        state1.dvar_M_South_SCADA := elit_Active;
        IF (("DB".state0.dvar_M_sup_South_Commands) = (elit_NoCommand)) THEN
            state1.dvar_M_sup_South_Commands := elit_DownstreamPaddleStop;
        ELSIF (("DB".state0.dvar_M_sup_South_Commands) = (elit_DownstreamGateOpen)) THEN
            state1.dvar_M_sup_South_Commands := elit_DownstreamGateOpen;
        ELSIF (("DB".state0.dvar_M_sup_South_Commands) = (elit_DownstreamGateClose)) THEN
            state1.dvar_M_sup_South_Commands := elit_DownstreamGateClose;
        ELSIF (("DB".state0.dvar_M_sup_South_Commands) = (elit_DownstreamGateStop)) THEN
            state1.dvar_M_sup_South_Commands := elit_DownstreamGateStop;
        ELSIF (("DB".state0.dvar_M_sup_South_Commands) = (elit_DownstreamPaddleOpen)) THEN
            state1.dvar_M_sup_South_Commands := elit_DownstreamPaddleOpen;
        ELSIF (("DB".state0.dvar_M_sup_South_Commands) = (elit_DownstreamPaddleClose)) THEN
            state1.dvar_M_sup_South_Commands := elit_DownstreamPaddleClose;
        ELSIF (("DB".state0.dvar_M_sup_South_Commands) = (elit_DownstreamPaddleStop)) THEN
            state1.dvar_M_sup_South_Commands := elit_DownstreamPaddleStop;
        ELSIF (("DB".state0.dvar_M_sup_South_Commands) = (elit_DownstreamEnteringTLRedRed)) THEN
            state1.dvar_M_sup_South_Commands := elit_DownstreamEnteringTLRedRed;
        ELSIF (("DB".state0.dvar_M_sup_South_Commands) = (elit_DownstreamEnteringTLRed)) THEN
            state1.dvar_M_sup_South_Commands := elit_DownstreamEnteringTLRed;
        ELSIF (("DB".state0.dvar_M_sup_South_Commands) = (elit_DownstreamEnteringTLRedGreen)) THEN
            state1.dvar_M_sup_South_Commands := elit_DownstreamEnteringTLRedGreen;
        ELSIF (("DB".state0.dvar_M_sup_South_Commands) = (elit_DownstreamEnteringTLGreen)) THEN
            state1.dvar_M_sup_South_Commands := elit_DownstreamEnteringTLGreen;
        ELSIF (("DB".state0.dvar_M_sup_South_Commands) = (elit_DownstreamLeavingTLRed)) THEN
            state1.dvar_M_sup_South_Commands := elit_DownstreamLeavingTLRed;
        ELSIF (("DB".state0.dvar_M_sup_South_Commands) = (elit_DownstreamLeavingTLGreen)) THEN
            state1.dvar_M_sup_South_Commands := elit_DownstreamLeavingTLGreen;
        ELSIF (("DB".state0.dvar_M_sup_South_Commands) = (elit_UpstreamGateOpen)) THEN
            state1.dvar_M_sup_South_Commands := elit_UpstreamGateOpen;
        ELSIF (("DB".state0.dvar_M_sup_South_Commands) = (elit_UpstreamGateClose)) THEN
            state1.dvar_M_sup_South_Commands := elit_UpstreamGateClose;
        ELSIF (("DB".state0.dvar_M_sup_South_Commands) = (elit_UpstreamGateStop)) THEN
            state1.dvar_M_sup_South_Commands := elit_UpstreamGateStop;
        ELSIF (("DB".state0.dvar_M_sup_South_Commands) = (elit_UpstreamPaddleOpen)) THEN
            state1.dvar_M_sup_South_Commands := elit_UpstreamPaddleOpen;
        ELSIF (("DB".state0.dvar_M_sup_South_Commands) = (elit_UpstreamPaddleClose)) THEN
            state1.dvar_M_sup_South_Commands := elit_UpstreamPaddleClose;
        ELSIF (("DB".state0.dvar_M_sup_South_Commands) = (elit_UpstreamPaddleStop)) THEN
            state1.dvar_M_sup_South_Commands := elit_UpstreamPaddleStop;
        ELSIF (("DB".state0.dvar_M_sup_South_Commands) = (elit_UpstreamEnteringTLRedRed)) THEN
            state1.dvar_M_sup_South_Commands := elit_UpstreamEnteringTLRedRed;
        ELSIF (("DB".state0.dvar_M_sup_South_Commands) = (elit_UpstreamEnteringTLRed)) THEN
            state1.dvar_M_sup_South_Commands := elit_UpstreamEnteringTLRed;
        ELSIF (("DB".state0.dvar_M_sup_South_Commands) = (elit_UpstreamEnteringTLRedGreen)) THEN
            state1.dvar_M_sup_South_Commands := elit_UpstreamEnteringTLRedGreen;
        ELSIF (("DB".state0.dvar_M_sup_South_Commands) = (elit_UpstreamEnteringTLGreen)) THEN
            state1.dvar_M_sup_South_Commands := elit_UpstreamEnteringTLGreen;
        ELSIF (("DB".state0.dvar_M_sup_South_Commands) = (elit_UpstreamLeavingTLRed)) THEN
            state1.dvar_M_sup_South_Commands := elit_UpstreamLeavingTLRed;
        ELSIF (("DB".state0.dvar_M_sup_South_Commands) = (elit_UpstreamLeavingTLGreen)) THEN
            state1.dvar_M_sup_South_Commands := elit_UpstreamLeavingTLGreen;
        END_IF;

        "DB".state0 := state1;
    END_IF;
END_IF;

// Event "South_Commands_UpstreamEnteringTLGreen_act".
IF NOT progress THEN
    b1 := ("DB".state0.dvar_M_South_SCADA) = (elit_Inactive);
    b1 := b1 AND ("SCADA".dvar_M_South_SCADA_UpstreamEnteringTLGreen);
    IF b1 THEN
        progress := TRUE;
        state1 := "DB".state0;

        state1.dvar_M_South_SCADA := elit_Active;
        IF (("DB".state0.dvar_M_sup_South_Commands) = (elit_NoCommand)) THEN
            state1.dvar_M_sup_South_Commands := elit_UpstreamEnteringTLGreen;
        ELSIF (("DB".state0.dvar_M_sup_South_Commands) = (elit_DownstreamGateOpen)) THEN
            state1.dvar_M_sup_South_Commands := elit_DownstreamGateOpen;
        ELSIF (("DB".state0.dvar_M_sup_South_Commands) = (elit_DownstreamGateClose)) THEN
            state1.dvar_M_sup_South_Commands := elit_DownstreamGateClose;
        ELSIF (("DB".state0.dvar_M_sup_South_Commands) = (elit_DownstreamGateStop)) THEN
            state1.dvar_M_sup_South_Commands := elit_DownstreamGateStop;
        ELSIF (("DB".state0.dvar_M_sup_South_Commands) = (elit_DownstreamPaddleOpen)) THEN
            state1.dvar_M_sup_South_Commands := elit_DownstreamPaddleOpen;
        ELSIF (("DB".state0.dvar_M_sup_South_Commands) = (elit_DownstreamPaddleClose)) THEN
            state1.dvar_M_sup_South_Commands := elit_DownstreamPaddleClose;
        ELSIF (("DB".state0.dvar_M_sup_South_Commands) = (elit_DownstreamPaddleStop)) THEN
            state1.dvar_M_sup_South_Commands := elit_DownstreamPaddleStop;
        ELSIF (("DB".state0.dvar_M_sup_South_Commands) = (elit_DownstreamEnteringTLRedRed)) THEN
            state1.dvar_M_sup_South_Commands := elit_DownstreamEnteringTLRedRed;
        ELSIF (("DB".state0.dvar_M_sup_South_Commands) = (elit_DownstreamEnteringTLRed)) THEN
            state1.dvar_M_sup_South_Commands := elit_DownstreamEnteringTLRed;
        ELSIF (("DB".state0.dvar_M_sup_South_Commands) = (elit_DownstreamEnteringTLRedGreen)) THEN
            state1.dvar_M_sup_South_Commands := elit_DownstreamEnteringTLRedGreen;
        ELSIF (("DB".state0.dvar_M_sup_South_Commands) = (elit_DownstreamEnteringTLGreen)) THEN
            state1.dvar_M_sup_South_Commands := elit_DownstreamEnteringTLGreen;
        ELSIF (("DB".state0.dvar_M_sup_South_Commands) = (elit_DownstreamLeavingTLRed)) THEN
            state1.dvar_M_sup_South_Commands := elit_DownstreamLeavingTLRed;
        ELSIF (("DB".state0.dvar_M_sup_South_Commands) = (elit_DownstreamLeavingTLGreen)) THEN
            state1.dvar_M_sup_South_Commands := elit_DownstreamLeavingTLGreen;
        ELSIF (("DB".state0.dvar_M_sup_South_Commands) = (elit_UpstreamGateOpen)) THEN
            state1.dvar_M_sup_South_Commands := elit_UpstreamGateOpen;
        ELSIF (("DB".state0.dvar_M_sup_South_Commands) = (elit_UpstreamGateClose)) THEN
            state1.dvar_M_sup_South_Commands := elit_UpstreamGateClose;
        ELSIF (("DB".state0.dvar_M_sup_South_Commands) = (elit_UpstreamGateStop)) THEN
            state1.dvar_M_sup_South_Commands := elit_UpstreamGateStop;
        ELSIF (("DB".state0.dvar_M_sup_South_Commands) = (elit_UpstreamPaddleOpen)) THEN
            state1.dvar_M_sup_South_Commands := elit_UpstreamPaddleOpen;
        ELSIF (("DB".state0.dvar_M_sup_South_Commands) = (elit_UpstreamPaddleClose)) THEN
            state1.dvar_M_sup_South_Commands := elit_UpstreamPaddleClose;
        ELSIF (("DB".state0.dvar_M_sup_South_Commands) = (elit_UpstreamPaddleStop)) THEN
            state1.dvar_M_sup_South_Commands := elit_UpstreamPaddleStop;
        ELSIF (("DB".state0.dvar_M_sup_South_Commands) = (elit_UpstreamEnteringTLRedRed)) THEN
            state1.dvar_M_sup_South_Commands := elit_UpstreamEnteringTLRedRed;
        ELSIF (("DB".state0.dvar_M_sup_South_Commands) = (elit_UpstreamEnteringTLRed)) THEN
            state1.dvar_M_sup_South_Commands := elit_UpstreamEnteringTLRed;
        ELSIF (("DB".state0.dvar_M_sup_South_Commands) = (elit_UpstreamEnteringTLRedGreen)) THEN
            state1.dvar_M_sup_South_Commands := elit_UpstreamEnteringTLRedGreen;
        ELSIF (("DB".state0.dvar_M_sup_South_Commands) = (elit_UpstreamEnteringTLGreen)) THEN
            state1.dvar_M_sup_South_Commands := elit_UpstreamEnteringTLGreen;
        ELSIF (("DB".state0.dvar_M_sup_South_Commands) = (elit_UpstreamLeavingTLRed)) THEN
            state1.dvar_M_sup_South_Commands := elit_UpstreamLeavingTLRed;
        ELSIF (("DB".state0.dvar_M_sup_South_Commands) = (elit_UpstreamLeavingTLGreen)) THEN
            state1.dvar_M_sup_South_Commands := elit_UpstreamLeavingTLGreen;
        END_IF;

        "DB".state0 := state1;
    END_IF;
END_IF;

// Event "South_Commands_UpstreamEnteringTLRed_act".
IF NOT progress THEN
    b1 := ("DB".state0.dvar_M_South_SCADA) = (elit_Inactive);
    b1 := b1 AND ("SCADA".dvar_M_South_SCADA_UpstreamEnteringTLRed);
    IF b1 THEN
        progress := TRUE;
        state1 := "DB".state0;

        state1.dvar_M_South_SCADA := elit_Active;
        IF (("DB".state0.dvar_M_sup_South_Commands) = (elit_NoCommand)) THEN
            state1.dvar_M_sup_South_Commands := elit_UpstreamEnteringTLRed;
        ELSIF (("DB".state0.dvar_M_sup_South_Commands) = (elit_DownstreamGateOpen)) THEN
            state1.dvar_M_sup_South_Commands := elit_DownstreamGateOpen;
        ELSIF (("DB".state0.dvar_M_sup_South_Commands) = (elit_DownstreamGateClose)) THEN
            state1.dvar_M_sup_South_Commands := elit_DownstreamGateClose;
        ELSIF (("DB".state0.dvar_M_sup_South_Commands) = (elit_DownstreamGateStop)) THEN
            state1.dvar_M_sup_South_Commands := elit_DownstreamGateStop;
        ELSIF (("DB".state0.dvar_M_sup_South_Commands) = (elit_DownstreamPaddleOpen)) THEN
            state1.dvar_M_sup_South_Commands := elit_DownstreamPaddleOpen;
        ELSIF (("DB".state0.dvar_M_sup_South_Commands) = (elit_DownstreamPaddleClose)) THEN
            state1.dvar_M_sup_South_Commands := elit_DownstreamPaddleClose;
        ELSIF (("DB".state0.dvar_M_sup_South_Commands) = (elit_DownstreamPaddleStop)) THEN
            state1.dvar_M_sup_South_Commands := elit_DownstreamPaddleStop;
        ELSIF (("DB".state0.dvar_M_sup_South_Commands) = (elit_DownstreamEnteringTLRedRed)) THEN
            state1.dvar_M_sup_South_Commands := elit_DownstreamEnteringTLRedRed;
        ELSIF (("DB".state0.dvar_M_sup_South_Commands) = (elit_DownstreamEnteringTLRed)) THEN
            state1.dvar_M_sup_South_Commands := elit_DownstreamEnteringTLRed;
        ELSIF (("DB".state0.dvar_M_sup_South_Commands) = (elit_DownstreamEnteringTLRedGreen)) THEN
            state1.dvar_M_sup_South_Commands := elit_DownstreamEnteringTLRedGreen;
        ELSIF (("DB".state0.dvar_M_sup_South_Commands) = (elit_DownstreamEnteringTLGreen)) THEN
            state1.dvar_M_sup_South_Commands := elit_DownstreamEnteringTLGreen;
        ELSIF (("DB".state0.dvar_M_sup_South_Commands) = (elit_DownstreamLeavingTLRed)) THEN
            state1.dvar_M_sup_South_Commands := elit_DownstreamLeavingTLRed;
        ELSIF (("DB".state0.dvar_M_sup_South_Commands) = (elit_DownstreamLeavingTLGreen)) THEN
            state1.dvar_M_sup_South_Commands := elit_DownstreamLeavingTLGreen;
        ELSIF (("DB".state0.dvar_M_sup_South_Commands) = (elit_UpstreamGateOpen)) THEN
            state1.dvar_M_sup_South_Commands := elit_UpstreamGateOpen;
        ELSIF (("DB".state0.dvar_M_sup_South_Commands) = (elit_UpstreamGateClose)) THEN
            state1.dvar_M_sup_South_Commands := elit_UpstreamGateClose;
        ELSIF (("DB".state0.dvar_M_sup_South_Commands) = (elit_UpstreamGateStop)) THEN
            state1.dvar_M_sup_South_Commands := elit_UpstreamGateStop;
        ELSIF (("DB".state0.dvar_M_sup_South_Commands) = (elit_UpstreamPaddleOpen)) THEN
            state1.dvar_M_sup_South_Commands := elit_UpstreamPaddleOpen;
        ELSIF (("DB".state0.dvar_M_sup_South_Commands) = (elit_UpstreamPaddleClose)) THEN
            state1.dvar_M_sup_South_Commands := elit_UpstreamPaddleClose;
        ELSIF (("DB".state0.dvar_M_sup_South_Commands) = (elit_UpstreamPaddleStop)) THEN
            state1.dvar_M_sup_South_Commands := elit_UpstreamPaddleStop;
        ELSIF (("DB".state0.dvar_M_sup_South_Commands) = (elit_UpstreamEnteringTLRedRed)) THEN
            state1.dvar_M_sup_South_Commands := elit_UpstreamEnteringTLRedRed;
        ELSIF (("DB".state0.dvar_M_sup_South_Commands) = (elit_UpstreamEnteringTLRed)) THEN
            state1.dvar_M_sup_South_Commands := elit_UpstreamEnteringTLRed;
        ELSIF (("DB".state0.dvar_M_sup_South_Commands) = (elit_UpstreamEnteringTLRedGreen)) THEN
            state1.dvar_M_sup_South_Commands := elit_UpstreamEnteringTLRedGreen;
        ELSIF (("DB".state0.dvar_M_sup_South_Commands) = (elit_UpstreamEnteringTLGreen)) THEN
            state1.dvar_M_sup_South_Commands := elit_UpstreamEnteringTLGreen;
        ELSIF (("DB".state0.dvar_M_sup_South_Commands) = (elit_UpstreamLeavingTLRed)) THEN
            state1.dvar_M_sup_South_Commands := elit_UpstreamLeavingTLRed;
        ELSIF (("DB".state0.dvar_M_sup_South_Commands) = (elit_UpstreamLeavingTLGreen)) THEN
            state1.dvar_M_sup_South_Commands := elit_UpstreamLeavingTLGreen;
        END_IF;

        "DB".state0 := state1;
    END_IF;
END_IF;

// Event "South_Commands_UpstreamEnteringTLRedGreen_act".
IF NOT progress THEN
    b1 := ("DB".state0.dvar_M_South_SCADA) = (elit_Inactive);
    b1 := b1 AND ("SCADA".dvar_M_South_SCADA_UpstreamEnteringTLRedGreen);
    IF b1 THEN
        progress := TRUE;
        state1 := "DB".state0;

        state1.dvar_M_South_SCADA := elit_Active;
        IF (("DB".state0.dvar_M_sup_South_Commands) = (elit_NoCommand)) THEN
            state1.dvar_M_sup_South_Commands := elit_UpstreamEnteringTLRedGreen;
        ELSIF (("DB".state0.dvar_M_sup_South_Commands) = (elit_DownstreamGateOpen)) THEN
            state1.dvar_M_sup_South_Commands := elit_DownstreamGateOpen;
        ELSIF (("DB".state0.dvar_M_sup_South_Commands) = (elit_DownstreamGateClose)) THEN
            state1.dvar_M_sup_South_Commands := elit_DownstreamGateClose;
        ELSIF (("DB".state0.dvar_M_sup_South_Commands) = (elit_DownstreamGateStop)) THEN
            state1.dvar_M_sup_South_Commands := elit_DownstreamGateStop;
        ELSIF (("DB".state0.dvar_M_sup_South_Commands) = (elit_DownstreamPaddleOpen)) THEN
            state1.dvar_M_sup_South_Commands := elit_DownstreamPaddleOpen;
        ELSIF (("DB".state0.dvar_M_sup_South_Commands) = (elit_DownstreamPaddleClose)) THEN
            state1.dvar_M_sup_South_Commands := elit_DownstreamPaddleClose;
        ELSIF (("DB".state0.dvar_M_sup_South_Commands) = (elit_DownstreamPaddleStop)) THEN
            state1.dvar_M_sup_South_Commands := elit_DownstreamPaddleStop;
        ELSIF (("DB".state0.dvar_M_sup_South_Commands) = (elit_DownstreamEnteringTLRedRed)) THEN
            state1.dvar_M_sup_South_Commands := elit_DownstreamEnteringTLRedRed;
        ELSIF (("DB".state0.dvar_M_sup_South_Commands) = (elit_DownstreamEnteringTLRed)) THEN
            state1.dvar_M_sup_South_Commands := elit_DownstreamEnteringTLRed;
        ELSIF (("DB".state0.dvar_M_sup_South_Commands) = (elit_DownstreamEnteringTLRedGreen)) THEN
            state1.dvar_M_sup_South_Commands := elit_DownstreamEnteringTLRedGreen;
        ELSIF (("DB".state0.dvar_M_sup_South_Commands) = (elit_DownstreamEnteringTLGreen)) THEN
            state1.dvar_M_sup_South_Commands := elit_DownstreamEnteringTLGreen;
        ELSIF (("DB".state0.dvar_M_sup_South_Commands) = (elit_DownstreamLeavingTLRed)) THEN
            state1.dvar_M_sup_South_Commands := elit_DownstreamLeavingTLRed;
        ELSIF (("DB".state0.dvar_M_sup_South_Commands) = (elit_DownstreamLeavingTLGreen)) THEN
            state1.dvar_M_sup_South_Commands := elit_DownstreamLeavingTLGreen;
        ELSIF (("DB".state0.dvar_M_sup_South_Commands) = (elit_UpstreamGateOpen)) THEN
            state1.dvar_M_sup_South_Commands := elit_UpstreamGateOpen;
        ELSIF (("DB".state0.dvar_M_sup_South_Commands) = (elit_UpstreamGateClose)) THEN
            state1.dvar_M_sup_South_Commands := elit_UpstreamGateClose;
        ELSIF (("DB".state0.dvar_M_sup_South_Commands) = (elit_UpstreamGateStop)) THEN
            state1.dvar_M_sup_South_Commands := elit_UpstreamGateStop;
        ELSIF (("DB".state0.dvar_M_sup_South_Commands) = (elit_UpstreamPaddleOpen)) THEN
            state1.dvar_M_sup_South_Commands := elit_UpstreamPaddleOpen;
        ELSIF (("DB".state0.dvar_M_sup_South_Commands) = (elit_UpstreamPaddleClose)) THEN
            state1.dvar_M_sup_South_Commands := elit_UpstreamPaddleClose;
        ELSIF (("DB".state0.dvar_M_sup_South_Commands) = (elit_UpstreamPaddleStop)) THEN
            state1.dvar_M_sup_South_Commands := elit_UpstreamPaddleStop;
        ELSIF (("DB".state0.dvar_M_sup_South_Commands) = (elit_UpstreamEnteringTLRedRed)) THEN
            state1.dvar_M_sup_South_Commands := elit_UpstreamEnteringTLRedRed;
        ELSIF (("DB".state0.dvar_M_sup_South_Commands) = (elit_UpstreamEnteringTLRed)) THEN
            state1.dvar_M_sup_South_Commands := elit_UpstreamEnteringTLRed;
        ELSIF (("DB".state0.dvar_M_sup_South_Commands) = (elit_UpstreamEnteringTLRedGreen)) THEN
            state1.dvar_M_sup_South_Commands := elit_UpstreamEnteringTLRedGreen;
        ELSIF (("DB".state0.dvar_M_sup_South_Commands) = (elit_UpstreamEnteringTLGreen)) THEN
            state1.dvar_M_sup_South_Commands := elit_UpstreamEnteringTLGreen;
        ELSIF (("DB".state0.dvar_M_sup_South_Commands) = (elit_UpstreamLeavingTLRed)) THEN
            state1.dvar_M_sup_South_Commands := elit_UpstreamLeavingTLRed;
        ELSIF (("DB".state0.dvar_M_sup_South_Commands) = (elit_UpstreamLeavingTLGreen)) THEN
            state1.dvar_M_sup_South_Commands := elit_UpstreamLeavingTLGreen;
        END_IF;

        "DB".state0 := state1;
    END_IF;
END_IF;

// Event "South_Commands_UpstreamEnteringTLRedRed_act".
IF NOT progress THEN
    b1 := ("DB".state0.dvar_M_South_SCADA) = (elit_Inactive);
    b1 := b1 AND ("SCADA".dvar_M_South_SCADA_UpstreamEnteringTLRedRed);
    IF b1 THEN
        progress := TRUE;
        state1 := "DB".state0;

        state1.dvar_M_South_SCADA := elit_Active;
        IF (("DB".state0.dvar_M_sup_South_Commands) = (elit_NoCommand)) THEN
            state1.dvar_M_sup_South_Commands := elit_UpstreamEnteringTLRedRed;
        ELSIF (("DB".state0.dvar_M_sup_South_Commands) = (elit_DownstreamGateOpen)) THEN
            state1.dvar_M_sup_South_Commands := elit_DownstreamGateOpen;
        ELSIF (("DB".state0.dvar_M_sup_South_Commands) = (elit_DownstreamGateClose)) THEN
            state1.dvar_M_sup_South_Commands := elit_DownstreamGateClose;
        ELSIF (("DB".state0.dvar_M_sup_South_Commands) = (elit_DownstreamGateStop)) THEN
            state1.dvar_M_sup_South_Commands := elit_DownstreamGateStop;
        ELSIF (("DB".state0.dvar_M_sup_South_Commands) = (elit_DownstreamPaddleOpen)) THEN
            state1.dvar_M_sup_South_Commands := elit_DownstreamPaddleOpen;
        ELSIF (("DB".state0.dvar_M_sup_South_Commands) = (elit_DownstreamPaddleClose)) THEN
            state1.dvar_M_sup_South_Commands := elit_DownstreamPaddleClose;
        ELSIF (("DB".state0.dvar_M_sup_South_Commands) = (elit_DownstreamPaddleStop)) THEN
            state1.dvar_M_sup_South_Commands := elit_DownstreamPaddleStop;
        ELSIF (("DB".state0.dvar_M_sup_South_Commands) = (elit_DownstreamEnteringTLRedRed)) THEN
            state1.dvar_M_sup_South_Commands := elit_DownstreamEnteringTLRedRed;
        ELSIF (("DB".state0.dvar_M_sup_South_Commands) = (elit_DownstreamEnteringTLRed)) THEN
            state1.dvar_M_sup_South_Commands := elit_DownstreamEnteringTLRed;
        ELSIF (("DB".state0.dvar_M_sup_South_Commands) = (elit_DownstreamEnteringTLRedGreen)) THEN
            state1.dvar_M_sup_South_Commands := elit_DownstreamEnteringTLRedGreen;
        ELSIF (("DB".state0.dvar_M_sup_South_Commands) = (elit_DownstreamEnteringTLGreen)) THEN
            state1.dvar_M_sup_South_Commands := elit_DownstreamEnteringTLGreen;
        ELSIF (("DB".state0.dvar_M_sup_South_Commands) = (elit_DownstreamLeavingTLRed)) THEN
            state1.dvar_M_sup_South_Commands := elit_DownstreamLeavingTLRed;
        ELSIF (("DB".state0.dvar_M_sup_South_Commands) = (elit_DownstreamLeavingTLGreen)) THEN
            state1.dvar_M_sup_South_Commands := elit_DownstreamLeavingTLGreen;
        ELSIF (("DB".state0.dvar_M_sup_South_Commands) = (elit_UpstreamGateOpen)) THEN
            state1.dvar_M_sup_South_Commands := elit_UpstreamGateOpen;
        ELSIF (("DB".state0.dvar_M_sup_South_Commands) = (elit_UpstreamGateClose)) THEN
            state1.dvar_M_sup_South_Commands := elit_UpstreamGateClose;
        ELSIF (("DB".state0.dvar_M_sup_South_Commands) = (elit_UpstreamGateStop)) THEN
            state1.dvar_M_sup_South_Commands := elit_UpstreamGateStop;
        ELSIF (("DB".state0.dvar_M_sup_South_Commands) = (elit_UpstreamPaddleOpen)) THEN
            state1.dvar_M_sup_South_Commands := elit_UpstreamPaddleOpen;
        ELSIF (("DB".state0.dvar_M_sup_South_Commands) = (elit_UpstreamPaddleClose)) THEN
            state1.dvar_M_sup_South_Commands := elit_UpstreamPaddleClose;
        ELSIF (("DB".state0.dvar_M_sup_South_Commands) = (elit_UpstreamPaddleStop)) THEN
            state1.dvar_M_sup_South_Commands := elit_UpstreamPaddleStop;
        ELSIF (("DB".state0.dvar_M_sup_South_Commands) = (elit_UpstreamEnteringTLRedRed)) THEN
            state1.dvar_M_sup_South_Commands := elit_UpstreamEnteringTLRedRed;
        ELSIF (("DB".state0.dvar_M_sup_South_Commands) = (elit_UpstreamEnteringTLRed)) THEN
            state1.dvar_M_sup_South_Commands := elit_UpstreamEnteringTLRed;
        ELSIF (("DB".state0.dvar_M_sup_South_Commands) = (elit_UpstreamEnteringTLRedGreen)) THEN
            state1.dvar_M_sup_South_Commands := elit_UpstreamEnteringTLRedGreen;
        ELSIF (("DB".state0.dvar_M_sup_South_Commands) = (elit_UpstreamEnteringTLGreen)) THEN
            state1.dvar_M_sup_South_Commands := elit_UpstreamEnteringTLGreen;
        ELSIF (("DB".state0.dvar_M_sup_South_Commands) = (elit_UpstreamLeavingTLRed)) THEN
            state1.dvar_M_sup_South_Commands := elit_UpstreamLeavingTLRed;
        ELSIF (("DB".state0.dvar_M_sup_South_Commands) = (elit_UpstreamLeavingTLGreen)) THEN
            state1.dvar_M_sup_South_Commands := elit_UpstreamLeavingTLGreen;
        END_IF;

        "DB".state0 := state1;
    END_IF;
END_IF;

// Event "South_Commands_UpstreamGateClose_act".
IF NOT progress THEN
    b1 := ("DB".state0.dvar_M_South_SCADA) = (elit_Inactive);
    b1 := b1 AND ("SCADA".dvar_M_South_SCADA_UpstreamGateClose);
    IF b1 THEN
        progress := TRUE;
        state1 := "DB".state0;

        state1.dvar_M_South_SCADA := elit_Active;
        IF (("DB".state0.dvar_M_sup_South_Commands) = (elit_NoCommand)) THEN
            state1.dvar_M_sup_South_Commands := elit_UpstreamGateClose;
        ELSIF (("DB".state0.dvar_M_sup_South_Commands) = (elit_DownstreamGateOpen)) THEN
            state1.dvar_M_sup_South_Commands := elit_DownstreamGateOpen;
        ELSIF (("DB".state0.dvar_M_sup_South_Commands) = (elit_DownstreamGateClose)) THEN
            state1.dvar_M_sup_South_Commands := elit_DownstreamGateClose;
        ELSIF (("DB".state0.dvar_M_sup_South_Commands) = (elit_DownstreamGateStop)) THEN
            state1.dvar_M_sup_South_Commands := elit_DownstreamGateStop;
        ELSIF (("DB".state0.dvar_M_sup_South_Commands) = (elit_DownstreamPaddleOpen)) THEN
            state1.dvar_M_sup_South_Commands := elit_DownstreamPaddleOpen;
        ELSIF (("DB".state0.dvar_M_sup_South_Commands) = (elit_DownstreamPaddleClose)) THEN
            state1.dvar_M_sup_South_Commands := elit_DownstreamPaddleClose;
        ELSIF (("DB".state0.dvar_M_sup_South_Commands) = (elit_DownstreamPaddleStop)) THEN
            state1.dvar_M_sup_South_Commands := elit_DownstreamPaddleStop;
        ELSIF (("DB".state0.dvar_M_sup_South_Commands) = (elit_DownstreamEnteringTLRedRed)) THEN
            state1.dvar_M_sup_South_Commands := elit_DownstreamEnteringTLRedRed;
        ELSIF (("DB".state0.dvar_M_sup_South_Commands) = (elit_DownstreamEnteringTLRed)) THEN
            state1.dvar_M_sup_South_Commands := elit_DownstreamEnteringTLRed;
        ELSIF (("DB".state0.dvar_M_sup_South_Commands) = (elit_DownstreamEnteringTLRedGreen)) THEN
            state1.dvar_M_sup_South_Commands := elit_DownstreamEnteringTLRedGreen;
        ELSIF (("DB".state0.dvar_M_sup_South_Commands) = (elit_DownstreamEnteringTLGreen)) THEN
            state1.dvar_M_sup_South_Commands := elit_DownstreamEnteringTLGreen;
        ELSIF (("DB".state0.dvar_M_sup_South_Commands) = (elit_DownstreamLeavingTLRed)) THEN
            state1.dvar_M_sup_South_Commands := elit_DownstreamLeavingTLRed;
        ELSIF (("DB".state0.dvar_M_sup_South_Commands) = (elit_DownstreamLeavingTLGreen)) THEN
            state1.dvar_M_sup_South_Commands := elit_DownstreamLeavingTLGreen;
        ELSIF (("DB".state0.dvar_M_sup_South_Commands) = (elit_UpstreamGateOpen)) THEN
            state1.dvar_M_sup_South_Commands := elit_UpstreamGateOpen;
        ELSIF (("DB".state0.dvar_M_sup_South_Commands) = (elit_UpstreamGateClose)) THEN
            state1.dvar_M_sup_South_Commands := elit_UpstreamGateClose;
        ELSIF (("DB".state0.dvar_M_sup_South_Commands) = (elit_UpstreamGateStop)) THEN
            state1.dvar_M_sup_South_Commands := elit_UpstreamGateStop;
        ELSIF (("DB".state0.dvar_M_sup_South_Commands) = (elit_UpstreamPaddleOpen)) THEN
            state1.dvar_M_sup_South_Commands := elit_UpstreamPaddleOpen;
        ELSIF (("DB".state0.dvar_M_sup_South_Commands) = (elit_UpstreamPaddleClose)) THEN
            state1.dvar_M_sup_South_Commands := elit_UpstreamPaddleClose;
        ELSIF (("DB".state0.dvar_M_sup_South_Commands) = (elit_UpstreamPaddleStop)) THEN
            state1.dvar_M_sup_South_Commands := elit_UpstreamPaddleStop;
        ELSIF (("DB".state0.dvar_M_sup_South_Commands) = (elit_UpstreamEnteringTLRedRed)) THEN
            state1.dvar_M_sup_South_Commands := elit_UpstreamEnteringTLRedRed;
        ELSIF (("DB".state0.dvar_M_sup_South_Commands) = (elit_UpstreamEnteringTLRed)) THEN
            state1.dvar_M_sup_South_Commands := elit_UpstreamEnteringTLRed;
        ELSIF (("DB".state0.dvar_M_sup_South_Commands) = (elit_UpstreamEnteringTLRedGreen)) THEN
            state1.dvar_M_sup_South_Commands := elit_UpstreamEnteringTLRedGreen;
        ELSIF (("DB".state0.dvar_M_sup_South_Commands) = (elit_UpstreamEnteringTLGreen)) THEN
            state1.dvar_M_sup_South_Commands := elit_UpstreamEnteringTLGreen;
        ELSIF (("DB".state0.dvar_M_sup_South_Commands) = (elit_UpstreamLeavingTLRed)) THEN
            state1.dvar_M_sup_South_Commands := elit_UpstreamLeavingTLRed;
        ELSIF (("DB".state0.dvar_M_sup_South_Commands) = (elit_UpstreamLeavingTLGreen)) THEN
            state1.dvar_M_sup_South_Commands := elit_UpstreamLeavingTLGreen;
        END_IF;

        "DB".state0 := state1;
    END_IF;
END_IF;

// Event "South_Commands_UpstreamGateOpen_act".
IF NOT progress THEN
    b1 := ("DB".state0.dvar_M_South_SCADA) = (elit_Inactive);
    b1 := b1 AND ("SCADA".dvar_M_South_SCADA_UpstreamGateOpen);
    IF b1 THEN
        progress := TRUE;
        state1 := "DB".state0;

        state1.dvar_M_South_SCADA := elit_Active;
        IF (("DB".state0.dvar_M_sup_South_Commands) = (elit_NoCommand)) THEN
            state1.dvar_M_sup_South_Commands := elit_UpstreamGateOpen;
        ELSIF (("DB".state0.dvar_M_sup_South_Commands) = (elit_DownstreamGateOpen)) THEN
            state1.dvar_M_sup_South_Commands := elit_DownstreamGateOpen;
        ELSIF (("DB".state0.dvar_M_sup_South_Commands) = (elit_DownstreamGateClose)) THEN
            state1.dvar_M_sup_South_Commands := elit_DownstreamGateClose;
        ELSIF (("DB".state0.dvar_M_sup_South_Commands) = (elit_DownstreamGateStop)) THEN
            state1.dvar_M_sup_South_Commands := elit_DownstreamGateStop;
        ELSIF (("DB".state0.dvar_M_sup_South_Commands) = (elit_DownstreamPaddleOpen)) THEN
            state1.dvar_M_sup_South_Commands := elit_DownstreamPaddleOpen;
        ELSIF (("DB".state0.dvar_M_sup_South_Commands) = (elit_DownstreamPaddleClose)) THEN
            state1.dvar_M_sup_South_Commands := elit_DownstreamPaddleClose;
        ELSIF (("DB".state0.dvar_M_sup_South_Commands) = (elit_DownstreamPaddleStop)) THEN
            state1.dvar_M_sup_South_Commands := elit_DownstreamPaddleStop;
        ELSIF (("DB".state0.dvar_M_sup_South_Commands) = (elit_DownstreamEnteringTLRedRed)) THEN
            state1.dvar_M_sup_South_Commands := elit_DownstreamEnteringTLRedRed;
        ELSIF (("DB".state0.dvar_M_sup_South_Commands) = (elit_DownstreamEnteringTLRed)) THEN
            state1.dvar_M_sup_South_Commands := elit_DownstreamEnteringTLRed;
        ELSIF (("DB".state0.dvar_M_sup_South_Commands) = (elit_DownstreamEnteringTLRedGreen)) THEN
            state1.dvar_M_sup_South_Commands := elit_DownstreamEnteringTLRedGreen;
        ELSIF (("DB".state0.dvar_M_sup_South_Commands) = (elit_DownstreamEnteringTLGreen)) THEN
            state1.dvar_M_sup_South_Commands := elit_DownstreamEnteringTLGreen;
        ELSIF (("DB".state0.dvar_M_sup_South_Commands) = (elit_DownstreamLeavingTLRed)) THEN
            state1.dvar_M_sup_South_Commands := elit_DownstreamLeavingTLRed;
        ELSIF (("DB".state0.dvar_M_sup_South_Commands) = (elit_DownstreamLeavingTLGreen)) THEN
            state1.dvar_M_sup_South_Commands := elit_DownstreamLeavingTLGreen;
        ELSIF (("DB".state0.dvar_M_sup_South_Commands) = (elit_UpstreamGateOpen)) THEN
            state1.dvar_M_sup_South_Commands := elit_UpstreamGateOpen;
        ELSIF (("DB".state0.dvar_M_sup_South_Commands) = (elit_UpstreamGateClose)) THEN
            state1.dvar_M_sup_South_Commands := elit_UpstreamGateClose;
        ELSIF (("DB".state0.dvar_M_sup_South_Commands) = (elit_UpstreamGateStop)) THEN
            state1.dvar_M_sup_South_Commands := elit_UpstreamGateStop;
        ELSIF (("DB".state0.dvar_M_sup_South_Commands) = (elit_UpstreamPaddleOpen)) THEN
            state1.dvar_M_sup_South_Commands := elit_UpstreamPaddleOpen;
        ELSIF (("DB".state0.dvar_M_sup_South_Commands) = (elit_UpstreamPaddleClose)) THEN
            state1.dvar_M_sup_South_Commands := elit_UpstreamPaddleClose;
        ELSIF (("DB".state0.dvar_M_sup_South_Commands) = (elit_UpstreamPaddleStop)) THEN
            state1.dvar_M_sup_South_Commands := elit_UpstreamPaddleStop;
        ELSIF (("DB".state0.dvar_M_sup_South_Commands) = (elit_UpstreamEnteringTLRedRed)) THEN
            state1.dvar_M_sup_South_Commands := elit_UpstreamEnteringTLRedRed;
        ELSIF (("DB".state0.dvar_M_sup_South_Commands) = (elit_UpstreamEnteringTLRed)) THEN
            state1.dvar_M_sup_South_Commands := elit_UpstreamEnteringTLRed;
        ELSIF (("DB".state0.dvar_M_sup_South_Commands) = (elit_UpstreamEnteringTLRedGreen)) THEN
            state1.dvar_M_sup_South_Commands := elit_UpstreamEnteringTLRedGreen;
        ELSIF (("DB".state0.dvar_M_sup_South_Commands) = (elit_UpstreamEnteringTLGreen)) THEN
            state1.dvar_M_sup_South_Commands := elit_UpstreamEnteringTLGreen;
        ELSIF (("DB".state0.dvar_M_sup_South_Commands) = (elit_UpstreamLeavingTLRed)) THEN
            state1.dvar_M_sup_South_Commands := elit_UpstreamLeavingTLRed;
        ELSIF (("DB".state0.dvar_M_sup_South_Commands) = (elit_UpstreamLeavingTLGreen)) THEN
            state1.dvar_M_sup_South_Commands := elit_UpstreamLeavingTLGreen;
        END_IF;

        "DB".state0 := state1;
    END_IF;
END_IF;

// Event "South_Commands_UpstreamGateStop_act".
IF NOT progress THEN
    b1 := ("DB".state0.dvar_M_South_SCADA) = (elit_Inactive);
    b1 := b1 AND ("SCADA".dvar_M_South_SCADA_UpstreamGateStop);
    IF b1 THEN
        progress := TRUE;
        state1 := "DB".state0;

        state1.dvar_M_South_SCADA := elit_Active;
        IF (("DB".state0.dvar_M_sup_South_Commands) = (elit_NoCommand)) THEN
            state1.dvar_M_sup_South_Commands := elit_UpstreamGateStop;
        ELSIF (("DB".state0.dvar_M_sup_South_Commands) = (elit_DownstreamGateOpen)) THEN
            state1.dvar_M_sup_South_Commands := elit_DownstreamGateOpen;
        ELSIF (("DB".state0.dvar_M_sup_South_Commands) = (elit_DownstreamGateClose)) THEN
            state1.dvar_M_sup_South_Commands := elit_DownstreamGateClose;
        ELSIF (("DB".state0.dvar_M_sup_South_Commands) = (elit_DownstreamGateStop)) THEN
            state1.dvar_M_sup_South_Commands := elit_DownstreamGateStop;
        ELSIF (("DB".state0.dvar_M_sup_South_Commands) = (elit_DownstreamPaddleOpen)) THEN
            state1.dvar_M_sup_South_Commands := elit_DownstreamPaddleOpen;
        ELSIF (("DB".state0.dvar_M_sup_South_Commands) = (elit_DownstreamPaddleClose)) THEN
            state1.dvar_M_sup_South_Commands := elit_DownstreamPaddleClose;
        ELSIF (("DB".state0.dvar_M_sup_South_Commands) = (elit_DownstreamPaddleStop)) THEN
            state1.dvar_M_sup_South_Commands := elit_DownstreamPaddleStop;
        ELSIF (("DB".state0.dvar_M_sup_South_Commands) = (elit_DownstreamEnteringTLRedRed)) THEN
            state1.dvar_M_sup_South_Commands := elit_DownstreamEnteringTLRedRed;
        ELSIF (("DB".state0.dvar_M_sup_South_Commands) = (elit_DownstreamEnteringTLRed)) THEN
            state1.dvar_M_sup_South_Commands := elit_DownstreamEnteringTLRed;
        ELSIF (("DB".state0.dvar_M_sup_South_Commands) = (elit_DownstreamEnteringTLRedGreen)) THEN
            state1.dvar_M_sup_South_Commands := elit_DownstreamEnteringTLRedGreen;
        ELSIF (("DB".state0.dvar_M_sup_South_Commands) = (elit_DownstreamEnteringTLGreen)) THEN
            state1.dvar_M_sup_South_Commands := elit_DownstreamEnteringTLGreen;
        ELSIF (("DB".state0.dvar_M_sup_South_Commands) = (elit_DownstreamLeavingTLRed)) THEN
            state1.dvar_M_sup_South_Commands := elit_DownstreamLeavingTLRed;
        ELSIF (("DB".state0.dvar_M_sup_South_Commands) = (elit_DownstreamLeavingTLGreen)) THEN
            state1.dvar_M_sup_South_Commands := elit_DownstreamLeavingTLGreen;
        ELSIF (("DB".state0.dvar_M_sup_South_Commands) = (elit_UpstreamGateOpen)) THEN
            state1.dvar_M_sup_South_Commands := elit_UpstreamGateOpen;
        ELSIF (("DB".state0.dvar_M_sup_South_Commands) = (elit_UpstreamGateClose)) THEN
            state1.dvar_M_sup_South_Commands := elit_UpstreamGateClose;
        ELSIF (("DB".state0.dvar_M_sup_South_Commands) = (elit_UpstreamGateStop)) THEN
            state1.dvar_M_sup_South_Commands := elit_UpstreamGateStop;
        ELSIF (("DB".state0.dvar_M_sup_South_Commands) = (elit_UpstreamPaddleOpen)) THEN
            state1.dvar_M_sup_South_Commands := elit_UpstreamPaddleOpen;
        ELSIF (("DB".state0.dvar_M_sup_South_Commands) = (elit_UpstreamPaddleClose)) THEN
            state1.dvar_M_sup_South_Commands := elit_UpstreamPaddleClose;
        ELSIF (("DB".state0.dvar_M_sup_South_Commands) = (elit_UpstreamPaddleStop)) THEN
            state1.dvar_M_sup_South_Commands := elit_UpstreamPaddleStop;
        ELSIF (("DB".state0.dvar_M_sup_South_Commands) = (elit_UpstreamEnteringTLRedRed)) THEN
            state1.dvar_M_sup_South_Commands := elit_UpstreamEnteringTLRedRed;
        ELSIF (("DB".state0.dvar_M_sup_South_Commands) = (elit_UpstreamEnteringTLRed)) THEN
            state1.dvar_M_sup_South_Commands := elit_UpstreamEnteringTLRed;
        ELSIF (("DB".state0.dvar_M_sup_South_Commands) = (elit_UpstreamEnteringTLRedGreen)) THEN
            state1.dvar_M_sup_South_Commands := elit_UpstreamEnteringTLRedGreen;
        ELSIF (("DB".state0.dvar_M_sup_South_Commands) = (elit_UpstreamEnteringTLGreen)) THEN
            state1.dvar_M_sup_South_Commands := elit_UpstreamEnteringTLGreen;
        ELSIF (("DB".state0.dvar_M_sup_South_Commands) = (elit_UpstreamLeavingTLRed)) THEN
            state1.dvar_M_sup_South_Commands := elit_UpstreamLeavingTLRed;
        ELSIF (("DB".state0.dvar_M_sup_South_Commands) = (elit_UpstreamLeavingTLGreen)) THEN
            state1.dvar_M_sup_South_Commands := elit_UpstreamLeavingTLGreen;
        END_IF;

        "DB".state0 := state1;
    END_IF;
END_IF;

// Event "South_Commands_UpstreamLeavingTLGreen_act".
IF NOT progress THEN
    b1 := ("DB".state0.dvar_M_South_SCADA) = (elit_Inactive);
    b1 := b1 AND ("SCADA".dvar_M_South_SCADA_UpstreamLeavingTLGreen);
    IF b1 THEN
        progress := TRUE;
        state1 := "DB".state0;

        state1.dvar_M_South_SCADA := elit_Active;
        IF (("DB".state0.dvar_M_sup_South_Commands) = (elit_NoCommand)) THEN
            state1.dvar_M_sup_South_Commands := elit_UpstreamLeavingTLGreen;
        ELSIF (("DB".state0.dvar_M_sup_South_Commands) = (elit_DownstreamGateOpen)) THEN
            state1.dvar_M_sup_South_Commands := elit_DownstreamGateOpen;
        ELSIF (("DB".state0.dvar_M_sup_South_Commands) = (elit_DownstreamGateClose)) THEN
            state1.dvar_M_sup_South_Commands := elit_DownstreamGateClose;
        ELSIF (("DB".state0.dvar_M_sup_South_Commands) = (elit_DownstreamGateStop)) THEN
            state1.dvar_M_sup_South_Commands := elit_DownstreamGateStop;
        ELSIF (("DB".state0.dvar_M_sup_South_Commands) = (elit_DownstreamPaddleOpen)) THEN
            state1.dvar_M_sup_South_Commands := elit_DownstreamPaddleOpen;
        ELSIF (("DB".state0.dvar_M_sup_South_Commands) = (elit_DownstreamPaddleClose)) THEN
            state1.dvar_M_sup_South_Commands := elit_DownstreamPaddleClose;
        ELSIF (("DB".state0.dvar_M_sup_South_Commands) = (elit_DownstreamPaddleStop)) THEN
            state1.dvar_M_sup_South_Commands := elit_DownstreamPaddleStop;
        ELSIF (("DB".state0.dvar_M_sup_South_Commands) = (elit_DownstreamEnteringTLRedRed)) THEN
            state1.dvar_M_sup_South_Commands := elit_DownstreamEnteringTLRedRed;
        ELSIF (("DB".state0.dvar_M_sup_South_Commands) = (elit_DownstreamEnteringTLRed)) THEN
            state1.dvar_M_sup_South_Commands := elit_DownstreamEnteringTLRed;
        ELSIF (("DB".state0.dvar_M_sup_South_Commands) = (elit_DownstreamEnteringTLRedGreen)) THEN
            state1.dvar_M_sup_South_Commands := elit_DownstreamEnteringTLRedGreen;
        ELSIF (("DB".state0.dvar_M_sup_South_Commands) = (elit_DownstreamEnteringTLGreen)) THEN
            state1.dvar_M_sup_South_Commands := elit_DownstreamEnteringTLGreen;
        ELSIF (("DB".state0.dvar_M_sup_South_Commands) = (elit_DownstreamLeavingTLRed)) THEN
            state1.dvar_M_sup_South_Commands := elit_DownstreamLeavingTLRed;
        ELSIF (("DB".state0.dvar_M_sup_South_Commands) = (elit_DownstreamLeavingTLGreen)) THEN
            state1.dvar_M_sup_South_Commands := elit_DownstreamLeavingTLGreen;
        ELSIF (("DB".state0.dvar_M_sup_South_Commands) = (elit_UpstreamGateOpen)) THEN
            state1.dvar_M_sup_South_Commands := elit_UpstreamGateOpen;
        ELSIF (("DB".state0.dvar_M_sup_South_Commands) = (elit_UpstreamGateClose)) THEN
            state1.dvar_M_sup_South_Commands := elit_UpstreamGateClose;
        ELSIF (("DB".state0.dvar_M_sup_South_Commands) = (elit_UpstreamGateStop)) THEN
            state1.dvar_M_sup_South_Commands := elit_UpstreamGateStop;
        ELSIF (("DB".state0.dvar_M_sup_South_Commands) = (elit_UpstreamPaddleOpen)) THEN
            state1.dvar_M_sup_South_Commands := elit_UpstreamPaddleOpen;
        ELSIF (("DB".state0.dvar_M_sup_South_Commands) = (elit_UpstreamPaddleClose)) THEN
            state1.dvar_M_sup_South_Commands := elit_UpstreamPaddleClose;
        ELSIF (("DB".state0.dvar_M_sup_South_Commands) = (elit_UpstreamPaddleStop)) THEN
            state1.dvar_M_sup_South_Commands := elit_UpstreamPaddleStop;
        ELSIF (("DB".state0.dvar_M_sup_South_Commands) = (elit_UpstreamEnteringTLRedRed)) THEN
            state1.dvar_M_sup_South_Commands := elit_UpstreamEnteringTLRedRed;
        ELSIF (("DB".state0.dvar_M_sup_South_Commands) = (elit_UpstreamEnteringTLRed)) THEN
            state1.dvar_M_sup_South_Commands := elit_UpstreamEnteringTLRed;
        ELSIF (("DB".state0.dvar_M_sup_South_Commands) = (elit_UpstreamEnteringTLRedGreen)) THEN
            state1.dvar_M_sup_South_Commands := elit_UpstreamEnteringTLRedGreen;
        ELSIF (("DB".state0.dvar_M_sup_South_Commands) = (elit_UpstreamEnteringTLGreen)) THEN
            state1.dvar_M_sup_South_Commands := elit_UpstreamEnteringTLGreen;
        ELSIF (("DB".state0.dvar_M_sup_South_Commands) = (elit_UpstreamLeavingTLRed)) THEN
            state1.dvar_M_sup_South_Commands := elit_UpstreamLeavingTLRed;
        ELSIF (("DB".state0.dvar_M_sup_South_Commands) = (elit_UpstreamLeavingTLGreen)) THEN
            state1.dvar_M_sup_South_Commands := elit_UpstreamLeavingTLGreen;
        END_IF;

        "DB".state0 := state1;
    END_IF;
END_IF;

// Event "South_Commands_UpstreamLeavingTLRed_act".
IF NOT progress THEN
    b1 := ("DB".state0.dvar_M_South_SCADA) = (elit_Inactive);
    b1 := b1 AND ("SCADA".dvar_M_South_SCADA_UpstreamLeavingTLRed);
    IF b1 THEN
        progress := TRUE;
        state1 := "DB".state0;

        state1.dvar_M_South_SCADA := elit_Active;
        IF (("DB".state0.dvar_M_sup_South_Commands) = (elit_NoCommand)) THEN
            state1.dvar_M_sup_South_Commands := elit_UpstreamLeavingTLRed;
        ELSIF (("DB".state0.dvar_M_sup_South_Commands) = (elit_DownstreamGateOpen)) THEN
            state1.dvar_M_sup_South_Commands := elit_DownstreamGateOpen;
        ELSIF (("DB".state0.dvar_M_sup_South_Commands) = (elit_DownstreamGateClose)) THEN
            state1.dvar_M_sup_South_Commands := elit_DownstreamGateClose;
        ELSIF (("DB".state0.dvar_M_sup_South_Commands) = (elit_DownstreamGateStop)) THEN
            state1.dvar_M_sup_South_Commands := elit_DownstreamGateStop;
        ELSIF (("DB".state0.dvar_M_sup_South_Commands) = (elit_DownstreamPaddleOpen)) THEN
            state1.dvar_M_sup_South_Commands := elit_DownstreamPaddleOpen;
        ELSIF (("DB".state0.dvar_M_sup_South_Commands) = (elit_DownstreamPaddleClose)) THEN
            state1.dvar_M_sup_South_Commands := elit_DownstreamPaddleClose;
        ELSIF (("DB".state0.dvar_M_sup_South_Commands) = (elit_DownstreamPaddleStop)) THEN
            state1.dvar_M_sup_South_Commands := elit_DownstreamPaddleStop;
        ELSIF (("DB".state0.dvar_M_sup_South_Commands) = (elit_DownstreamEnteringTLRedRed)) THEN
            state1.dvar_M_sup_South_Commands := elit_DownstreamEnteringTLRedRed;
        ELSIF (("DB".state0.dvar_M_sup_South_Commands) = (elit_DownstreamEnteringTLRed)) THEN
            state1.dvar_M_sup_South_Commands := elit_DownstreamEnteringTLRed;
        ELSIF (("DB".state0.dvar_M_sup_South_Commands) = (elit_DownstreamEnteringTLRedGreen)) THEN
            state1.dvar_M_sup_South_Commands := elit_DownstreamEnteringTLRedGreen;
        ELSIF (("DB".state0.dvar_M_sup_South_Commands) = (elit_DownstreamEnteringTLGreen)) THEN
            state1.dvar_M_sup_South_Commands := elit_DownstreamEnteringTLGreen;
        ELSIF (("DB".state0.dvar_M_sup_South_Commands) = (elit_DownstreamLeavingTLRed)) THEN
            state1.dvar_M_sup_South_Commands := elit_DownstreamLeavingTLRed;
        ELSIF (("DB".state0.dvar_M_sup_South_Commands) = (elit_DownstreamLeavingTLGreen)) THEN
            state1.dvar_M_sup_South_Commands := elit_DownstreamLeavingTLGreen;
        ELSIF (("DB".state0.dvar_M_sup_South_Commands) = (elit_UpstreamGateOpen)) THEN
            state1.dvar_M_sup_South_Commands := elit_UpstreamGateOpen;
        ELSIF (("DB".state0.dvar_M_sup_South_Commands) = (elit_UpstreamGateClose)) THEN
            state1.dvar_M_sup_South_Commands := elit_UpstreamGateClose;
        ELSIF (("DB".state0.dvar_M_sup_South_Commands) = (elit_UpstreamGateStop)) THEN
            state1.dvar_M_sup_South_Commands := elit_UpstreamGateStop;
        ELSIF (("DB".state0.dvar_M_sup_South_Commands) = (elit_UpstreamPaddleOpen)) THEN
            state1.dvar_M_sup_South_Commands := elit_UpstreamPaddleOpen;
        ELSIF (("DB".state0.dvar_M_sup_South_Commands) = (elit_UpstreamPaddleClose)) THEN
            state1.dvar_M_sup_South_Commands := elit_UpstreamPaddleClose;
        ELSIF (("DB".state0.dvar_M_sup_South_Commands) = (elit_UpstreamPaddleStop)) THEN
            state1.dvar_M_sup_South_Commands := elit_UpstreamPaddleStop;
        ELSIF (("DB".state0.dvar_M_sup_South_Commands) = (elit_UpstreamEnteringTLRedRed)) THEN
            state1.dvar_M_sup_South_Commands := elit_UpstreamEnteringTLRedRed;
        ELSIF (("DB".state0.dvar_M_sup_South_Commands) = (elit_UpstreamEnteringTLRed)) THEN
            state1.dvar_M_sup_South_Commands := elit_UpstreamEnteringTLRed;
        ELSIF (("DB".state0.dvar_M_sup_South_Commands) = (elit_UpstreamEnteringTLRedGreen)) THEN
            state1.dvar_M_sup_South_Commands := elit_UpstreamEnteringTLRedGreen;
        ELSIF (("DB".state0.dvar_M_sup_South_Commands) = (elit_UpstreamEnteringTLGreen)) THEN
            state1.dvar_M_sup_South_Commands := elit_UpstreamEnteringTLGreen;
        ELSIF (("DB".state0.dvar_M_sup_South_Commands) = (elit_UpstreamLeavingTLRed)) THEN
            state1.dvar_M_sup_South_Commands := elit_UpstreamLeavingTLRed;
        ELSIF (("DB".state0.dvar_M_sup_South_Commands) = (elit_UpstreamLeavingTLGreen)) THEN
            state1.dvar_M_sup_South_Commands := elit_UpstreamLeavingTLGreen;
        END_IF;

        "DB".state0 := state1;
    END_IF;
END_IF;

// Event "South_Commands_UpstreamPaddleClose_act".
IF NOT progress THEN
    b1 := ("DB".state0.dvar_M_South_SCADA) = (elit_Inactive);
    b1 := b1 AND ("SCADA".dvar_M_South_SCADA_UpstreamPaddleClose);
    IF b1 THEN
        progress := TRUE;
        state1 := "DB".state0;

        state1.dvar_M_South_SCADA := elit_Active;
        IF (("DB".state0.dvar_M_sup_South_Commands) = (elit_NoCommand)) THEN
            state1.dvar_M_sup_South_Commands := elit_UpstreamPaddleClose;
        ELSIF (("DB".state0.dvar_M_sup_South_Commands) = (elit_DownstreamGateOpen)) THEN
            state1.dvar_M_sup_South_Commands := elit_DownstreamGateOpen;
        ELSIF (("DB".state0.dvar_M_sup_South_Commands) = (elit_DownstreamGateClose)) THEN
            state1.dvar_M_sup_South_Commands := elit_DownstreamGateClose;
        ELSIF (("DB".state0.dvar_M_sup_South_Commands) = (elit_DownstreamGateStop)) THEN
            state1.dvar_M_sup_South_Commands := elit_DownstreamGateStop;
        ELSIF (("DB".state0.dvar_M_sup_South_Commands) = (elit_DownstreamPaddleOpen)) THEN
            state1.dvar_M_sup_South_Commands := elit_DownstreamPaddleOpen;
        ELSIF (("DB".state0.dvar_M_sup_South_Commands) = (elit_DownstreamPaddleClose)) THEN
            state1.dvar_M_sup_South_Commands := elit_DownstreamPaddleClose;
        ELSIF (("DB".state0.dvar_M_sup_South_Commands) = (elit_DownstreamPaddleStop)) THEN
            state1.dvar_M_sup_South_Commands := elit_DownstreamPaddleStop;
        ELSIF (("DB".state0.dvar_M_sup_South_Commands) = (elit_DownstreamEnteringTLRedRed)) THEN
            state1.dvar_M_sup_South_Commands := elit_DownstreamEnteringTLRedRed;
        ELSIF (("DB".state0.dvar_M_sup_South_Commands) = (elit_DownstreamEnteringTLRed)) THEN
            state1.dvar_M_sup_South_Commands := elit_DownstreamEnteringTLRed;
        ELSIF (("DB".state0.dvar_M_sup_South_Commands) = (elit_DownstreamEnteringTLRedGreen)) THEN
            state1.dvar_M_sup_South_Commands := elit_DownstreamEnteringTLRedGreen;
        ELSIF (("DB".state0.dvar_M_sup_South_Commands) = (elit_DownstreamEnteringTLGreen)) THEN
            state1.dvar_M_sup_South_Commands := elit_DownstreamEnteringTLGreen;
        ELSIF (("DB".state0.dvar_M_sup_South_Commands) = (elit_DownstreamLeavingTLRed)) THEN
            state1.dvar_M_sup_South_Commands := elit_DownstreamLeavingTLRed;
        ELSIF (("DB".state0.dvar_M_sup_South_Commands) = (elit_DownstreamLeavingTLGreen)) THEN
            state1.dvar_M_sup_South_Commands := elit_DownstreamLeavingTLGreen;
        ELSIF (("DB".state0.dvar_M_sup_South_Commands) = (elit_UpstreamGateOpen)) THEN
            state1.dvar_M_sup_South_Commands := elit_UpstreamGateOpen;
        ELSIF (("DB".state0.dvar_M_sup_South_Commands) = (elit_UpstreamGateClose)) THEN
            state1.dvar_M_sup_South_Commands := elit_UpstreamGateClose;
        ELSIF (("DB".state0.dvar_M_sup_South_Commands) = (elit_UpstreamGateStop)) THEN
            state1.dvar_M_sup_South_Commands := elit_UpstreamGateStop;
        ELSIF (("DB".state0.dvar_M_sup_South_Commands) = (elit_UpstreamPaddleOpen)) THEN
            state1.dvar_M_sup_South_Commands := elit_UpstreamPaddleOpen;
        ELSIF (("DB".state0.dvar_M_sup_South_Commands) = (elit_UpstreamPaddleClose)) THEN
            state1.dvar_M_sup_South_Commands := elit_UpstreamPaddleClose;
        ELSIF (("DB".state0.dvar_M_sup_South_Commands) = (elit_UpstreamPaddleStop)) THEN
            state1.dvar_M_sup_South_Commands := elit_UpstreamPaddleStop;
        ELSIF (("DB".state0.dvar_M_sup_South_Commands) = (elit_UpstreamEnteringTLRedRed)) THEN
            state1.dvar_M_sup_South_Commands := elit_UpstreamEnteringTLRedRed;
        ELSIF (("DB".state0.dvar_M_sup_South_Commands) = (elit_UpstreamEnteringTLRed)) THEN
            state1.dvar_M_sup_South_Commands := elit_UpstreamEnteringTLRed;
        ELSIF (("DB".state0.dvar_M_sup_South_Commands) = (elit_UpstreamEnteringTLRedGreen)) THEN
            state1.dvar_M_sup_South_Commands := elit_UpstreamEnteringTLRedGreen;
        ELSIF (("DB".state0.dvar_M_sup_South_Commands) = (elit_UpstreamEnteringTLGreen)) THEN
            state1.dvar_M_sup_South_Commands := elit_UpstreamEnteringTLGreen;
        ELSIF (("DB".state0.dvar_M_sup_South_Commands) = (elit_UpstreamLeavingTLRed)) THEN
            state1.dvar_M_sup_South_Commands := elit_UpstreamLeavingTLRed;
        ELSIF (("DB".state0.dvar_M_sup_South_Commands) = (elit_UpstreamLeavingTLGreen)) THEN
            state1.dvar_M_sup_South_Commands := elit_UpstreamLeavingTLGreen;
        END_IF;

        "DB".state0 := state1;
    END_IF;
END_IF;

// Event "South_Commands_UpstreamPaddleOpen_act".
IF NOT progress THEN
    b1 := ("DB".state0.dvar_M_South_SCADA) = (elit_Inactive);
    b1 := b1 AND ("SCADA".dvar_M_South_SCADA_UpstreamPaddleOpen);
    IF b1 THEN
        progress := TRUE;
        state1 := "DB".state0;

        state1.dvar_M_South_SCADA := elit_Active;
        IF (("DB".state0.dvar_M_sup_South_Commands) = (elit_NoCommand)) THEN
            state1.dvar_M_sup_South_Commands := elit_UpstreamPaddleOpen;
        ELSIF (("DB".state0.dvar_M_sup_South_Commands) = (elit_DownstreamGateOpen)) THEN
            state1.dvar_M_sup_South_Commands := elit_DownstreamGateOpen;
        ELSIF (("DB".state0.dvar_M_sup_South_Commands) = (elit_DownstreamGateClose)) THEN
            state1.dvar_M_sup_South_Commands := elit_DownstreamGateClose;
        ELSIF (("DB".state0.dvar_M_sup_South_Commands) = (elit_DownstreamGateStop)) THEN
            state1.dvar_M_sup_South_Commands := elit_DownstreamGateStop;
        ELSIF (("DB".state0.dvar_M_sup_South_Commands) = (elit_DownstreamPaddleOpen)) THEN
            state1.dvar_M_sup_South_Commands := elit_DownstreamPaddleOpen;
        ELSIF (("DB".state0.dvar_M_sup_South_Commands) = (elit_DownstreamPaddleClose)) THEN
            state1.dvar_M_sup_South_Commands := elit_DownstreamPaddleClose;
        ELSIF (("DB".state0.dvar_M_sup_South_Commands) = (elit_DownstreamPaddleStop)) THEN
            state1.dvar_M_sup_South_Commands := elit_DownstreamPaddleStop;
        ELSIF (("DB".state0.dvar_M_sup_South_Commands) = (elit_DownstreamEnteringTLRedRed)) THEN
            state1.dvar_M_sup_South_Commands := elit_DownstreamEnteringTLRedRed;
        ELSIF (("DB".state0.dvar_M_sup_South_Commands) = (elit_DownstreamEnteringTLRed)) THEN
            state1.dvar_M_sup_South_Commands := elit_DownstreamEnteringTLRed;
        ELSIF (("DB".state0.dvar_M_sup_South_Commands) = (elit_DownstreamEnteringTLRedGreen)) THEN
            state1.dvar_M_sup_South_Commands := elit_DownstreamEnteringTLRedGreen;
        ELSIF (("DB".state0.dvar_M_sup_South_Commands) = (elit_DownstreamEnteringTLGreen)) THEN
            state1.dvar_M_sup_South_Commands := elit_DownstreamEnteringTLGreen;
        ELSIF (("DB".state0.dvar_M_sup_South_Commands) = (elit_DownstreamLeavingTLRed)) THEN
            state1.dvar_M_sup_South_Commands := elit_DownstreamLeavingTLRed;
        ELSIF (("DB".state0.dvar_M_sup_South_Commands) = (elit_DownstreamLeavingTLGreen)) THEN
            state1.dvar_M_sup_South_Commands := elit_DownstreamLeavingTLGreen;
        ELSIF (("DB".state0.dvar_M_sup_South_Commands) = (elit_UpstreamGateOpen)) THEN
            state1.dvar_M_sup_South_Commands := elit_UpstreamGateOpen;
        ELSIF (("DB".state0.dvar_M_sup_South_Commands) = (elit_UpstreamGateClose)) THEN
            state1.dvar_M_sup_South_Commands := elit_UpstreamGateClose;
        ELSIF (("DB".state0.dvar_M_sup_South_Commands) = (elit_UpstreamGateStop)) THEN
            state1.dvar_M_sup_South_Commands := elit_UpstreamGateStop;
        ELSIF (("DB".state0.dvar_M_sup_South_Commands) = (elit_UpstreamPaddleOpen)) THEN
            state1.dvar_M_sup_South_Commands := elit_UpstreamPaddleOpen;
        ELSIF (("DB".state0.dvar_M_sup_South_Commands) = (elit_UpstreamPaddleClose)) THEN
            state1.dvar_M_sup_South_Commands := elit_UpstreamPaddleClose;
        ELSIF (("DB".state0.dvar_M_sup_South_Commands) = (elit_UpstreamPaddleStop)) THEN
            state1.dvar_M_sup_South_Commands := elit_UpstreamPaddleStop;
        ELSIF (("DB".state0.dvar_M_sup_South_Commands) = (elit_UpstreamEnteringTLRedRed)) THEN
            state1.dvar_M_sup_South_Commands := elit_UpstreamEnteringTLRedRed;
        ELSIF (("DB".state0.dvar_M_sup_South_Commands) = (elit_UpstreamEnteringTLRed)) THEN
            state1.dvar_M_sup_South_Commands := elit_UpstreamEnteringTLRed;
        ELSIF (("DB".state0.dvar_M_sup_South_Commands) = (elit_UpstreamEnteringTLRedGreen)) THEN
            state1.dvar_M_sup_South_Commands := elit_UpstreamEnteringTLRedGreen;
        ELSIF (("DB".state0.dvar_M_sup_South_Commands) = (elit_UpstreamEnteringTLGreen)) THEN
            state1.dvar_M_sup_South_Commands := elit_UpstreamEnteringTLGreen;
        ELSIF (("DB".state0.dvar_M_sup_South_Commands) = (elit_UpstreamLeavingTLRed)) THEN
            state1.dvar_M_sup_South_Commands := elit_UpstreamLeavingTLRed;
        ELSIF (("DB".state0.dvar_M_sup_South_Commands) = (elit_UpstreamLeavingTLGreen)) THEN
            state1.dvar_M_sup_South_Commands := elit_UpstreamLeavingTLGreen;
        END_IF;

        "DB".state0 := state1;
    END_IF;
END_IF;

// Event "South_Commands_UpstreamPaddleStop_act".
IF NOT progress THEN
    b1 := ("DB".state0.dvar_M_South_SCADA) = (elit_Inactive);
    b1 := b1 AND ("SCADA".dvar_M_South_SCADA_UpstreamPaddleStop);
    IF b1 THEN
        progress := TRUE;
        state1 := "DB".state0;

        state1.dvar_M_South_SCADA := elit_Active;
        IF (("DB".state0.dvar_M_sup_South_Commands) = (elit_NoCommand)) THEN
            state1.dvar_M_sup_South_Commands := elit_UpstreamPaddleStop;
        ELSIF (("DB".state0.dvar_M_sup_South_Commands) = (elit_DownstreamGateOpen)) THEN
            state1.dvar_M_sup_South_Commands := elit_DownstreamGateOpen;
        ELSIF (("DB".state0.dvar_M_sup_South_Commands) = (elit_DownstreamGateClose)) THEN
            state1.dvar_M_sup_South_Commands := elit_DownstreamGateClose;
        ELSIF (("DB".state0.dvar_M_sup_South_Commands) = (elit_DownstreamGateStop)) THEN
            state1.dvar_M_sup_South_Commands := elit_DownstreamGateStop;
        ELSIF (("DB".state0.dvar_M_sup_South_Commands) = (elit_DownstreamPaddleOpen)) THEN
            state1.dvar_M_sup_South_Commands := elit_DownstreamPaddleOpen;
        ELSIF (("DB".state0.dvar_M_sup_South_Commands) = (elit_DownstreamPaddleClose)) THEN
            state1.dvar_M_sup_South_Commands := elit_DownstreamPaddleClose;
        ELSIF (("DB".state0.dvar_M_sup_South_Commands) = (elit_DownstreamPaddleStop)) THEN
            state1.dvar_M_sup_South_Commands := elit_DownstreamPaddleStop;
        ELSIF (("DB".state0.dvar_M_sup_South_Commands) = (elit_DownstreamEnteringTLRedRed)) THEN
            state1.dvar_M_sup_South_Commands := elit_DownstreamEnteringTLRedRed;
        ELSIF (("DB".state0.dvar_M_sup_South_Commands) = (elit_DownstreamEnteringTLRed)) THEN
            state1.dvar_M_sup_South_Commands := elit_DownstreamEnteringTLRed;
        ELSIF (("DB".state0.dvar_M_sup_South_Commands) = (elit_DownstreamEnteringTLRedGreen)) THEN
            state1.dvar_M_sup_South_Commands := elit_DownstreamEnteringTLRedGreen;
        ELSIF (("DB".state0.dvar_M_sup_South_Commands) = (elit_DownstreamEnteringTLGreen)) THEN
            state1.dvar_M_sup_South_Commands := elit_DownstreamEnteringTLGreen;
        ELSIF (("DB".state0.dvar_M_sup_South_Commands) = (elit_DownstreamLeavingTLRed)) THEN
            state1.dvar_M_sup_South_Commands := elit_DownstreamLeavingTLRed;
        ELSIF (("DB".state0.dvar_M_sup_South_Commands) = (elit_DownstreamLeavingTLGreen)) THEN
            state1.dvar_M_sup_South_Commands := elit_DownstreamLeavingTLGreen;
        ELSIF (("DB".state0.dvar_M_sup_South_Commands) = (elit_UpstreamGateOpen)) THEN
            state1.dvar_M_sup_South_Commands := elit_UpstreamGateOpen;
        ELSIF (("DB".state0.dvar_M_sup_South_Commands) = (elit_UpstreamGateClose)) THEN
            state1.dvar_M_sup_South_Commands := elit_UpstreamGateClose;
        ELSIF (("DB".state0.dvar_M_sup_South_Commands) = (elit_UpstreamGateStop)) THEN
            state1.dvar_M_sup_South_Commands := elit_UpstreamGateStop;
        ELSIF (("DB".state0.dvar_M_sup_South_Commands) = (elit_UpstreamPaddleOpen)) THEN
            state1.dvar_M_sup_South_Commands := elit_UpstreamPaddleOpen;
        ELSIF (("DB".state0.dvar_M_sup_South_Commands) = (elit_UpstreamPaddleClose)) THEN
            state1.dvar_M_sup_South_Commands := elit_UpstreamPaddleClose;
        ELSIF (("DB".state0.dvar_M_sup_South_Commands) = (elit_UpstreamPaddleStop)) THEN
            state1.dvar_M_sup_South_Commands := elit_UpstreamPaddleStop;
        ELSIF (("DB".state0.dvar_M_sup_South_Commands) = (elit_UpstreamEnteringTLRedRed)) THEN
            state1.dvar_M_sup_South_Commands := elit_UpstreamEnteringTLRedRed;
        ELSIF (("DB".state0.dvar_M_sup_South_Commands) = (elit_UpstreamEnteringTLRed)) THEN
            state1.dvar_M_sup_South_Commands := elit_UpstreamEnteringTLRed;
        ELSIF (("DB".state0.dvar_M_sup_South_Commands) = (elit_UpstreamEnteringTLRedGreen)) THEN
            state1.dvar_M_sup_South_Commands := elit_UpstreamEnteringTLRedGreen;
        ELSIF (("DB".state0.dvar_M_sup_South_Commands) = (elit_UpstreamEnteringTLGreen)) THEN
            state1.dvar_M_sup_South_Commands := elit_UpstreamEnteringTLGreen;
        ELSIF (("DB".state0.dvar_M_sup_South_Commands) = (elit_UpstreamLeavingTLRed)) THEN
            state1.dvar_M_sup_South_Commands := elit_UpstreamLeavingTLRed;
        ELSIF (("DB".state0.dvar_M_sup_South_Commands) = (elit_UpstreamLeavingTLGreen)) THEN
            state1.dvar_M_sup_South_Commands := elit_UpstreamLeavingTLGreen;
        END_IF;

        "DB".state0 := state1;
    END_IF;
END_IF;

// Event "South_Downstream_EnteringTLs_East_Actuator_c_g".
IF NOT progress THEN
    b1 := ("DB".state0.dvar_M_sup_South_Downstream_EnteringTLs_East_Actuator) = (elit_RedGreen);
    b1 := b1 AND (("DB".state0.dvar_M_sup_South_Downstream_LeavingTLs_East_Actuator) = (elit_Red));
    b1 := b1 AND (("DB".state0.dvar_M_sup_South_Downstream_LeavingTLs_East_SensorR) = (elit_On));
    b1 := b1 AND (("DB".state0.dvar_M_sup_South_Downstream_LeavingTLs_East_SensorG) = (elit_Off));
    b1 := b1 AND (("DB".state0.dvar_M_sup_South_Downstream_LeavingTLs_West_Actuator) = (elit_Red));
    b1 := b1 AND (("DB".state0.dvar_M_sup_South_Downstream_LeavingTLs_West_SensorR) = (elit_On));
    b1 := b1 AND (("DB".state0.dvar_M_sup_South_Downstream_LeavingTLs_West_SensorG) = (elit_Off));
    b1 := b1 AND (("DB".state0.dvar_M_sup_South_Downstream_Gates_East_Actuator) = (elit_Rest));
    b1 := b1 AND (("DB".state0.dvar_M_sup_South_Downstream_Gates_East_Sensor) = (elit_Open));
    b1 := b1 AND (("DB".state0.dvar_M_sup_South_Downstream_Gates_West_Actuator) = (elit_Rest));
    b1 := b1 AND (("DB".state0.dvar_M_sup_South_Downstream_Gates_West_Sensor) = (elit_Open));
    b1 := b1 AND (("DB".state0.dvar_M_sup_South_Commands) = (elit_DownstreamEnteringTLGreen));
    IF b1 THEN
        progress := TRUE;
        state1 := "DB".state0;

        state1.dvar_M_South_HW_EnteringTL_BNH_East_Q_Green := TRUE;
        state1.dvar_M_sup_South_Downstream_EnteringTLs_East_Actuator := elit_Green;

        "DB".state0 := state1;
    END_IF;
END_IF;

// Event "South_Downstream_EnteringTLs_East_Actuator_c_r".
IF NOT progress THEN
    b2 := ("DB".state0.dvar_M_sup_South_Downstream_EnteringTLs_East_Actuator) = (elit_RedRed);
    b2 := b2 OR (("DB".state0.dvar_M_sup_South_Downstream_EnteringTLs_East_Actuator) = (elit_RedGreen));
    b2 := b2 OR (("DB".state0.dvar_M_sup_South_Downstream_EnteringTLs_East_Actuator) = (elit_Green));
    b1 := b2;
    b1 := b1 AND (("DB".state0.dvar_M_sup_South_Commands) = (elit_DownstreamEnteringTLRed));
    IF b1 THEN
        progress := TRUE;
        state1 := "DB".state0;

        state1.dvar_M_South_HW_EnteringTL_BNH_East_Q_Red := TRUE;
        state1.dvar_M_South_HW_EnteringTL_BNH_East_Q_Green := FALSE;
        state1.dvar_M_South_HW_EnteringTL_BNH_East_Q_RedRed := FALSE;
        IF (("DB".state0.dvar_M_sup_South_Downstream_EnteringTLs_East_Actuator) = (elit_RedRed)) THEN
            state1.dvar_M_sup_South_Downstream_EnteringTLs_East_Actuator := elit_Red;
        ELSIF (("DB".state0.dvar_M_sup_South_Downstream_EnteringTLs_East_Actuator) = (elit_RedGreen)) THEN
            state1.dvar_M_sup_South_Downstream_EnteringTLs_East_Actuator := elit_Red;
        ELSIF (("DB".state0.dvar_M_sup_South_Downstream_EnteringTLs_East_Actuator) = (elit_Green)) THEN
            state1.dvar_M_sup_South_Downstream_EnteringTLs_East_Actuator := elit_Red;
        END_IF;

        "DB".state0 := state1;
    END_IF;
END_IF;

// Event "South_Downstream_EnteringTLs_East_Actuator_c_rg".
IF NOT progress THEN
    b1 := ("DB".state0.dvar_M_sup_South_Downstream_EnteringTLs_East_Actuator) = (elit_Red);
    b1 := b1 AND (("DB".state0.dvar_M_sup_South_Commands) = (elit_DownstreamEnteringTLRedGreen));
    IF b1 THEN
        progress := TRUE;
        state1 := "DB".state0;

        state1.dvar_M_South_HW_EnteringTL_BNH_East_Q_Red := TRUE;
        state1.dvar_M_South_HW_EnteringTL_BNH_East_Q_Green := TRUE;
        state1.dvar_M_sup_South_Downstream_EnteringTLs_East_Actuator := elit_RedGreen;

        "DB".state0 := state1;
    END_IF;
END_IF;

// Event "South_Downstream_EnteringTLs_East_Actuator_c_rr".
IF NOT progress THEN
    b1 := ("DB".state0.dvar_M_sup_South_Downstream_EnteringTLs_East_Actuator) = (elit_Red);
    b1 := b1 AND (("DB".state0.dvar_M_sup_South_Commands) = (elit_DownstreamEnteringTLRedRed));
    IF b1 THEN
        progress := TRUE;
        state1 := "DB".state0;

        state1.dvar_M_South_HW_EnteringTL_BNH_East_Q_RedRed := TRUE;
        state1.dvar_M_sup_South_Downstream_EnteringTLs_East_Actuator := elit_RedRed;

        "DB".state0 := state1;
    END_IF;
END_IF;

// Event "South_Downstream_EnteringTLs_East_SensorG_u_off".
IF NOT progress THEN
    b1 := NOT(ivar_M_South_HW_EnteringTL_BNH_East_Green);
    IF b1 THEN
        b2 := ("DB".state0.dvar_M_sup_South_Downstream_EnteringTLs_East_Actuator) = (elit_Red);
        b2 := b2 OR (("DB".state0.dvar_M_sup_South_Downstream_EnteringTLs_East_Actuator) = (elit_RedRed));
        b1 := b1 AND (b2);
    END_IF;
    b1 := b1 AND (("DB".state0.dvar_M_sup_South_Downstream_EnteringTLs_East_SensorG) = (elit_On));
    IF b1 THEN
        progress := TRUE;
        state1 := "DB".state0;

        state1.dvar_M_sup_South_Downstream_EnteringTLs_East_SensorG := elit_Off;

        "DB".state0 := state1;
    END_IF;
END_IF;
END_FUNCTION
